{attribute 'qualified_only'}
{attribute 'strict'}
{attribute 'to_string'}
// Default CHAN 1, add 0x800 next channel
TYPE E_Module :
(
    CHAN1	:= 1,
    CHAN2	:= 2,
    CHAN3	:= 3
) WORD;
END_TYPE

(* stored: Version 1.1.0.1
   DUT E_Module: Id {09bbb0a9-83d3-4934-a810-426e9d69fb51} *)
